// TIA Portal V19 export
TYPE "LAF_typeAxisDiagWarningWord"
TITLE = LAF_typeAxisDiagWarningWord
// Warnings of a Technology Object
// stored: Access Published
   STRUCT
      bit00_SystemWarning { ExternalWritable := 'False'} : Bool;   // A system-internal error has occurred / Enable
      bit01_ConfigWarning { ExternalWritable := 'False'} : Bool;   // Configuration error. One or several configuration parameters are adjusted internally / Error
      bit02_UserWarning { ExternalWritable := 'False'} : Bool;   // Error in user program at a Motion Control instruction or its use / RestartActive
      bit03_CommandNotAccepted { ExternalWritable := 'False'} : Bool;   // Job cannot be executed. A Motion Control instruction cannot be executed because the necessary conditions have not been met / OnlineStartValuesChanged
      bit04_DriveWarning { ExternalWritable := 'False'} : Bool;   // Warning of the drive. When a warning message is pending at the drive that does not result in a TO alarm, this bit is not set. Evaluate the drive warnings directly using the status word of the drive / ControlPanelActive
      bit05_SensorWarning { ExternalWritable := 'False'} : Bool;   // Error in encoder system / HomingDone
      bit06_DynamicWarning { ExternalWritable := 'False'} : Bool;   // Specified dynamic values are limited to permissible values / Done
      bit07_CommunicationWarning { ExternalWritable := 'False'} : Bool;   // Communication error. Missing or faulty communication. / StandStill
      bit08_SWLimitMin { ExternalWritable := 'False'} : Bool;   // The negative software limit switch has been approached / PositioningCommand
      bit09_SWLimitMax { ExternalWritable := 'False'} : Bool;   // The positive software limit switch has been approached / JogCommand
      bit10_HomingWarning { ExternalWritable := 'False'} : Bool;   // Error during homing operation. The homing cannot be completed / VelocityCommand
      bit11_FollowingErrorWarning { ExternalWritable := 'False'} : Bool;   // Warning limit of following error monitoring reached/exceeded / HomingCommand
      bit12_PositioningWarning { ExternalWritable := 'False'} : Bool;   // Positioning error / ConstantVelocity
      bit13_PeripheralWarning { ExternalWritable := 'False'} : Bool;   // Error accessing a logical address / Accelerating
      bit14_SynchronousWarning { ExternalWritable := 'False'} : Bool;   // Error during synchronous operation. The leading axis specified in the Motion Control instruction was not configured as a possible leading axis / Decelerating
      bit15_AdaptionWarning { ExternalWritable := 'False'} : Bool;   // Error in automatic data transfer / SWLimitMinActive
      bit16_Reserved { ExternalWritable := 'False'} : Bool;   // Reserved / SWLimitMaxActive
      bit17_Reserved { ExternalWritable := 'False'} : Bool;   // Reserved / HWLimitMinActive
      bit18_Reserved { ExternalWritable := 'False'} : Bool;   // Reserved / HWLimitMaxActive
      bit19_Reserved { ExternalWritable := 'False'} : Bool;   // Reserved
      bit20_Reserved { ExternalWritable := 'False'} : Bool;   // Reserved
      bit21_Reserved { ExternalWritable := 'False'} : Bool;   // Reserved / Synchronizing
      bit22_Reserved { ExternalWritable := 'False'} : Bool;   // Reserved / Synhronous
      bit23_Reserved { ExternalWritable := 'False'} : Bool;   // Reserved / SuperimposedMotionCommand
      bit24_Reserved { ExternalWritable := 'False'} : Bool;   // Reserved / PhasingCommand
      bit25_Reserved { ExternalWritable := 'False'} : Bool;   // Reserved / AxisSimulation
      bit26_Reserved { ExternalWritable := 'False'} : Bool;   // Reserved / TorqueLimitingCommand
      bit27_Reserved { ExternalWritable := 'False'} : Bool;   // Reserved / InLimitation
      bit28_Reserved { ExternalWritable := 'False'} : Bool;   // Reserved / NonPositionControlled
      bit29_Reserved { ExternalWritable := 'False'} : Bool;   // Reserved
      bit30_Reserved { ExternalWritable := 'False'} : Bool;   // Reserved / InClamping
      bit31_Reserved { ExternalWritable := 'False'} : Bool;   // Reserved
   END_STRUCT;
END_TYPE
